(* IEC 61131-3 sources: industrial-digital-twin/openplc-programs, 3 files *)

(* ---- barrier.st ---- *)
PROGRAM BarrierControl
VAR
    // Входы от Java модели (через Modbus)
    OpenCmd AT %IX0.0 : BOOL;      // Команда открыть
    CloseCmd AT %IX0.1 : BOOL;     // Команда закрыть

    // Выходы на Java модель
    Angle AT %QW0 : INT;            // Угол стрелы (0-900 = 0-90°)
    LimitOpen AT %QX0.0 : BOOL;     // Концевик открыт
    LimitClosed AT %QX0.1 : BOOL;   // Концевик закрыт
    Error AT %QX0.2 : BOOL;         // Флаг ошибки

    // Внутренние переменные
    currentAngle : INT := 0;
END_VAR

// Логика управления шлагбаумом
IF OpenCmd AND CloseCmd THEN
    // ОШИБКА: обе команды одновременно
    Error := TRUE;
    LimitOpen := FALSE;
    LimitClosed := FALSE;

ELSIF OpenCmd AND NOT Error THEN
    // Движение вверх
    IF currentAngle < 900 THEN
        currentAngle := currentAngle + 100;  // +10° за шаг
    END_IF;

    // Проверка концевика
    IF currentAngle >= 900 THEN
        currentAngle := 900;
        LimitOpen := TRUE;
        LimitClosed := FALSE;
    END_IF;

ELSIF CloseCmd AND NOT Error THEN
    // Движение вниз
    IF currentAngle > 0 THEN
        currentAngle := currentAngle - 100;  // -10° за шаг
    END_IF;

    // Проверка концевика
    IF currentAngle <= 0 THEN
        currentAngle := 0;
        LimitClosed := TRUE;
        LimitOpen := FALSE;
    END_IF;

ELSE
    // Нет ошибки, стоим на месте
    Error := FALSE;
END_IF;

// Запись угла на выход
Angle := currentAngle;
END_PROGRAM

// Конфигурация задач
TASK MainTask(INTERVAL := T#100ms, PRIORITY := 1);
PROGRAM INSTANCE BarrierControl WITH MainTask;
END_CONFIGURATION

(* ---- barrier_corrected.st ---- *)
// Программа управления шлагбаумом
// Угол меняется от 0 до 90 градусов

VAR_GLOBAL
    // Входные команды
    OpenCmd AT %IX0.0 : BOOL;      // Команда открыть
    CloseCmd AT %IX0.1 : BOOL;     // Команда закрыть

    // Выходные сигналы
    Angle AT %QW0 : INT;            // Текущий угол (0-900 = 0-90.0°)
    LimitOpen AT %QX0.0 : BOOL;     // Концевик открыт
    LimitClosed AT %QX0.1 : BOOL;   // Концевик закрыт
    ErrorFlag AT %QX0.2 : BOOL;     // Флаг ошибки
END_VAR

VAR
    currentAngle : INT := 0;
    lastOpenCmd : BOOL := FALSE;
    lastCloseCmd : BOOL := FALSE;
END_VAR

// Основная логика
// Проверка на одновременные команды
IF OpenCmd = TRUE AND CloseCmd = TRUE THEN
    ErrorFlag := TRUE;
    LimitOpen := FALSE;
    LimitClosed := FALSE;

ELSIF ErrorFlag = TRUE THEN
    // В ошибке - ничего не делаем
    // Нужен сброс перезагрузкой

ELSIF OpenCmd = TRUE AND lastOpenCmd = FALSE THEN
    // Открываем
    IF currentAngle < 900 THEN
        currentAngle := currentAngle + 100;
        LimitClosed := FALSE;
    END_IF;

    // Проверка концевика открыто
    IF currentAngle >= 900 THEN
        currentAngle := 900;
        LimitOpen := TRUE;
    END_IF;

    lastOpenCmd := TRUE;
    lastCloseCmd := FALSE;

ELSIF CloseCmd = TRUE AND lastCloseCmd = FALSE THEN
    // Закрываем
    IF currentAngle > 0 THEN
        currentAngle := currentAngle - 100;
        LimitOpen := FALSE;
    END_IF;

    // Проверка концевика закрыто
    IF currentAngle <= 0 THEN
        currentAngle := 0;
        LimitClosed := TRUE;
    END_IF;

    lastCloseCmd := TRUE;
    lastOpenCmd := FALSE;

ELSE
    // Обновляем последние команды
    lastOpenCmd := OpenCmd;
    lastCloseCmd := CloseCmd;
END_IF;

// Записываем угол на выход
Angle := currentAngle;

END_PROGRAM

// Конфигурация задачи
TASK Main(INTERVAL := T#100ms, PRIORITY := 1);
PROGRAM Instance WITH Main;
END_CONFIGURATION

(* ---- barrier_simple.st ---- *)
PROGRAM BarrierSimple
VAR
    OpenCmd AT %IX0.0 : BOOL;
    CloseCmd AT %IX0.1 : BOOL;
    Angle AT %QW0 : INT;
    LimitOpen AT %QX0.0 : BOOL;
    LimitClosed AT %QX0.1 : BOOL;
    Error AT %QX0.2 : BOOL;
    angle_val : INT := 0;
END_VAR

IF OpenCmd = TRUE AND CloseCmd = TRUE THEN
    Error := TRUE;
ELSIF OpenCmd = TRUE AND Error = FALSE THEN
    IF angle_val < 900 THEN
        angle_val := angle_val + 100;
    END_IF;
    LimitClosed := FALSE;
    IF angle_val >= 900 THEN
        angle_val := 900;
        LimitOpen := TRUE;
    END_IF;
ELSIF CloseCmd = TRUE AND Error = FALSE THEN
    IF angle_val > 0 THEN
        angle_val := angle_val - 100;
    END_IF;
    LimitOpen := FALSE;
    IF angle_val <= 0 THEN
        angle_val := 0;
        LimitClosed := TRUE;
    END_IF;
END_IF

Angle := angle_val;
END_PROGRAM

TASK Main(INTERVAL := T#100ms, PRIORITY := 1);
PROGRAM P1 WITH Main;
END_CONFIGURATION
